Xinje XCPPro project, PLC1: XC3-24 (software 3.3q)

PROGRAM Ladder

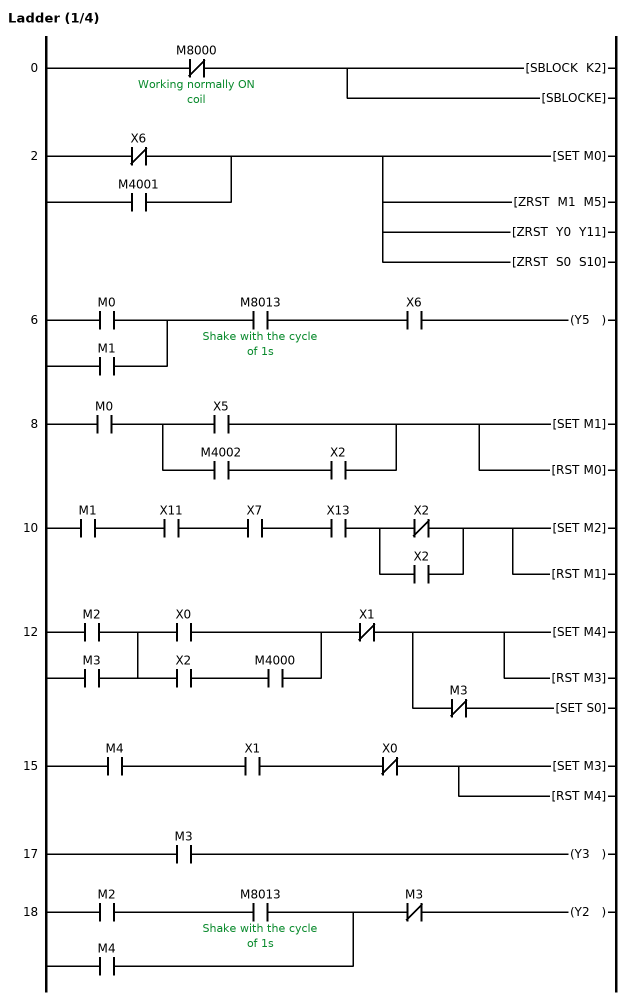
LDI    M8000	; Working normally ON coil
SBLOCK K2
SBLOCKE
LDI    X6
OR     M4001
SET    M0
ZRST   M1 M5
ZRST   Y0 Y11
ZRST   S0 S10
LD     M0
OR     M1
AND    M8013	; Shake with the cycle of 1s
AND    X6
OUT    Y5
LD     M0
LD     X5
LD     M4002
AND    X2
ORB
ANB
SET    M1
RST    M0
LD     M1
AND    X11
AND    X7
AND    X13
LDI    X2
OR     X2
ANB
SET    M2
RST    M1
LD     M2
OR     M3
LD     X0
LD     X2
AND    M4000
ORB
ANB
ANI    X1
SET    M4
RST    M3
ANI    M3
SET    S0
LD     M4
AND    X1
ANI    X0
SET    M3
RST    M4
LD     M3
OUT    Y3
LD     M2
AND    M8013	; Shake with the cycle of 1s
OR     M4
ANI    M3
OUT    Y2

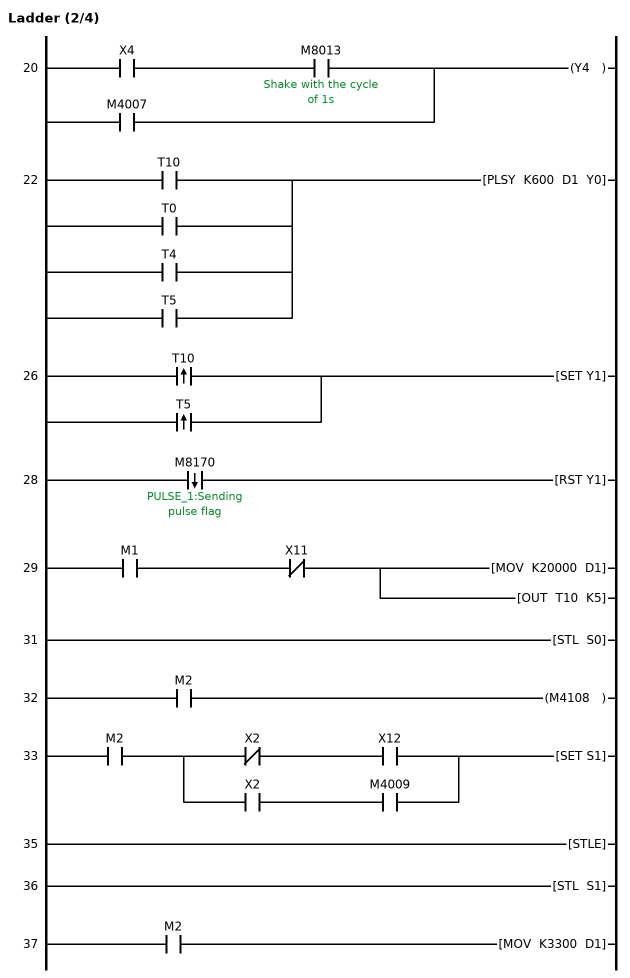
LD     X4
AND    M8013	; Shake with the cycle of 1s
OR     M4007
OUT    Y4
LD     T10
OR     T0
OR     T4
OR     T5
PLSY   K600 D1 Y0
LDP    T10
ORP    T5
SET    Y1
LDF    M8170	; PULSE_1:Sending pulse flag
RST    Y1
LD     M1
ANI    X11
MOV    K20000 D1
OUT    T10 K5
STL    S0
LD     M2
OUT    M4108
LD     M2
LDI    X2
AND    X12
LD     X2
AND    M4009
ORB
ANB
SET    S1
STLE
STL    S1
LD     M2
MOV    K3300 D1

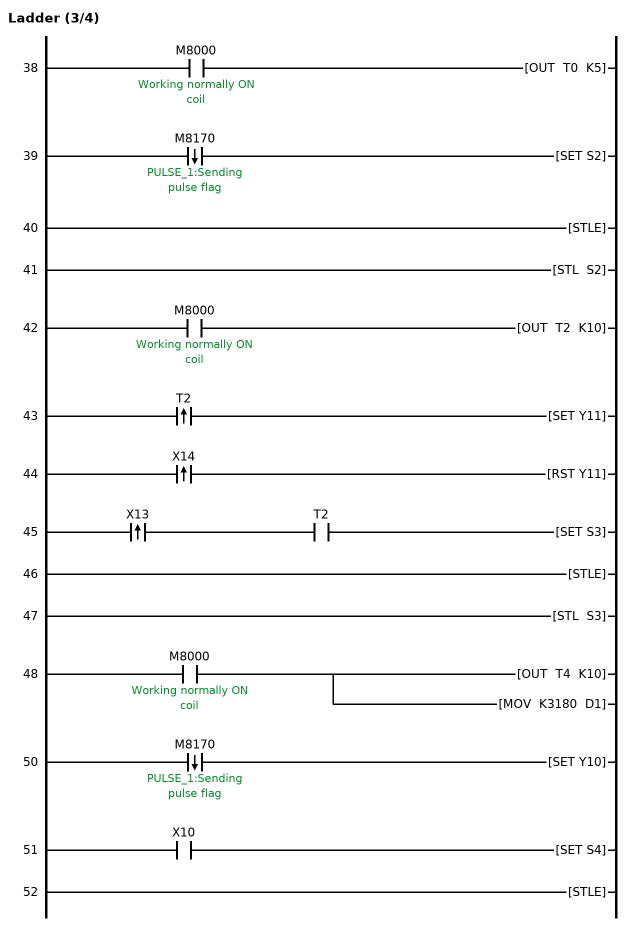
LD     M8000	; Working normally ON coil
OUT    T0 K5
LDF    M8170	; PULSE_1:Sending pulse flag
SET    S2
STLE
STL    S2
LD     M8000	; Working normally ON coil
OUT    T2 K10
LDP    T2
SET    Y11
LDP    X14
RST    Y11
LDP    X13
AND    T2
SET    S3
STLE
STL    S3
LD     M8000	; Working normally ON coil
OUT    T4 K10
MOV    K3180 D1
LDF    M8170	; PULSE_1:Sending pulse flag
SET    Y10
LD     X10
SET    S4
STLE

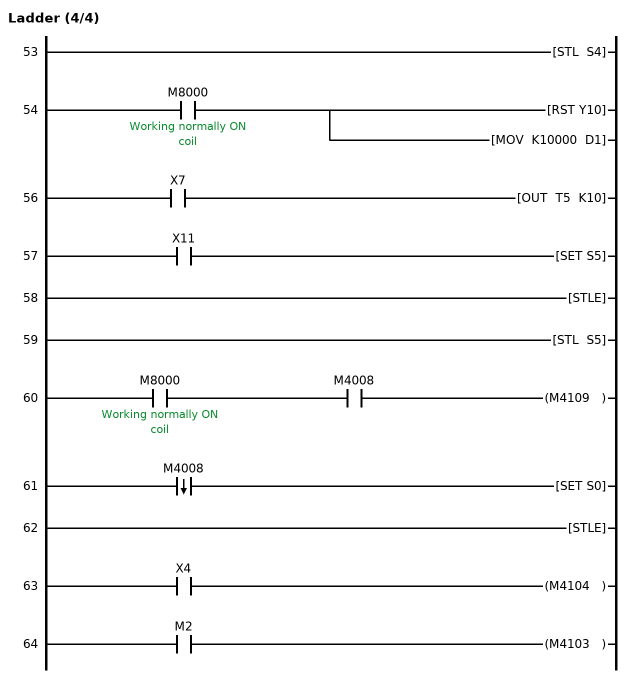
STL    S4
LD     M8000	; Working normally ON coil
RST    Y10
MOV    K10000 D1
LD     X7
OUT    T5 K10
LD     X11
SET    S5
STLE
STL    S5
LD     M8000	; Working normally ON coil
AND    M4008
OUT    M4109
LDF    M4008
SET    S0
STLE
LD     X4
OUT    M4104
LD     M2
OUT    M4103